Fanuc KAREL source: kt00739.KL

-- PROVISIONAL review KL for V1013-1; original PC SHA256 7ee263f555218975708955234a3025deb3b40a6eb1d1670db809ca628f6c3493
-- Incomplete behavior may be omitted. Consult companion uncertainty JSON. Do not deploy.
PROGRAM KT00739
%NOLOCKGROUP
VAR
  OUT : INTEGER
-- UNRESOLVED_DECL ARG type=002018
BEGIN
  -- UNRESOLVED_PC offsets 5-18; opcodes 22,1D,23
  -- UNRESOLVED_PC offsets 23-27; opcodes 7F
END KT00739
